TYPE (* Blink Marine PowerKey DI Struct *)
  (* Version 1.0, 2025-07-21, Franz Höpfinger, initial API and implementation and/or initial documentation *)
  PACKAGE BlinkMarine::io::DI;
  IMPORT eclipse4diac::core::TypeHash;
  PKP_2200_LI_DI_S : STRUCT
    Pin : USINT := 255;
  END_STRUCT;
END_TYPE
